// TwinCAT 3 PLC project CarlPlc
// ProgramVersion: 3.1.4022.1
// libraries:
//   Tc2_ModbusRTU, * (Beckhoff Automation GmbH)
//   Tc2_Standard, * (Beckhoff Automation GmbH)
//   Tc2_System, * (Beckhoff Automation GmbH)
//   Tc2_Utilities, * (Beckhoff Automation GmbH)
//   Tc3_Module, * (Beckhoff Automation GmbH)
// project tree:
//   Common/ DetectEvent.TcPOU (not stored), GVL_Common.TcGVL (not stored), TasterEventStates.TcDUT (not stored), TasterEventType.TcDUT (not stored), LinearCalibration.TcDUT (not stored)
//   FlowRateSensor/ GVL_FlowControl.TcGVL, PRG_UpdateFlowRateSensor.TcPOU (not stored)
//   GasAnalysis/ GVL_GasAnalysis.TcGVL (not stored), PRG_GasAnalysis.TcPOU (not stored)
//   GasSupply/ GVL_GasSupply.TcGVL (not stored), PRG_UpdateGasSupply.TcPOU (not stored)
//   MotorControl/ GVL_MotorControl.TcGVL (not stored), PRG_UpdateMotor.TcPOU
//   pHOrpControl/ EN_ModbusReadTarget.TcDUT, GVL_PhOrpControl.TcGVL (not stored), PRG_ReadModbusSensorData.TcPOU, PRG_UpdatePhControl.TcPOU
//   / PlcTask.TcTTO
//   MAIN/ MAIN.TcPOU
//   ReactorPressureControl/ GVL_ReactorPressureControl.TcGVL (not stored), PRG_UpdatePressureSensor.TcPOU (not stored)
//   RoomTempRh/ GVL_TempRHSensor.TcGVL (not stored), PRG_UpdateRoomTempRh.TcPOU
//   TemperatureControl/ EN_TempControlMode.TcDUT (not stored), FB_TON.TcPOU (not stored), GVL_TemperatureControl.TcGVL, FUN_ComputeMovingSetPoint.TcPOU (not stored), PRG_UpdateTemperatureControl.TcPOU (not stored), PRG_BAT_TemperatureControl.TcPOU
//   TemperatureControl/PID/ CLK_PRG.TcPOU (not stored), FB_PWM.TcPOU, FT_DERIV.TcPOU (not stored), FT_PIDWL.TcPOU (not stored), FT_PIWL.TcPOU (not stored), PWM_DC.TcPOU, TP_X.TcPOU (not stored), T_PLC_MS.TcPOU (not stored), T_PLC_US.TcPOU (not stored)
//   TemperatureControl/PID_Hoti/ FT_GET_GAINS.TcPOU, FT_PID_CAS.TcPOU, FT_PID_STERI.TcPOU, FT_P_J.TcPOU
// real-time tasks:
//   TASK PlcTask: cycle T#10ms, priority 20, ADS port 350
// I/O:
//   DEVICE Device 1 (EtherCAT), AmsNetId 5.54.16.198.2.1
//     Term 1 (EK1200) [EK1200-5000 EtherCAT Power supply (2A E-Bus)]
//       Term 2 (EL3014) Motor Speed In [EL3014 4Ch. Ana. Input 0-20mA DIFF]
//       Term 3 (EL4004) Motor Speed Out [EL4004 4Ch. Ana. Output 0-10V, 12bit]
//       Term 4 (EL2004) DO Heating Cooling [EL2004 4Ch. Dig. Output 24V, 0.5A]
//       Term 5 (EL2004) DO Gassing Valves [EL2004 4Ch. Dig. Output 24V, 0.5A]
//       Term 6 (EL2004) DO Motor Control Out [EL2004 4Ch. Dig. Output 24V, 0.5A]
//       Term 7 (EL6021) PhModbus [EL6021 Interface (RS422/485)]
//       Term 8 (EL6021) OrpModbus [EL6021 Interface (RS422/485)]
//       Term 21 (EL1004) DI Gas Analysis [EL1004 4Ch. Dig. Input 24V, 3ms]
//       Term 18 (EL3052) AI Pressure Flow [EL3052 2Ch. Ana. Input 4-20mA]
//       Term 24 (EL3052) AI Heating Cooling [EL3052 2Ch. Ana. Input 4-20mA]
//       Term 10 (EL9184) [EL9184 Potential Connection, 8 x 24V, 8 x Ground]
//       Term 26 (EL3044) [EL3044 4Ch. Ana. Input 0-20mA]
//       Term 9 (EL9011) [EL9011 End Terminal]
// variable links:
//   CarlPlc/CarlPlc Instance <-> Device 1 (EtherCAT)/Term 1 (EK1200)/Term 18 (EL3052) AI Pressure Flow
//     PlcTask Inputs/GVL_FlowControl.flowRateRawCounts <-> FlowRateSensor/FlowRateRaw
//     PlcTask Inputs/GVL_ReactorPressureControl.pressureRawCounts <-> PressureSensor/PressureSensorRaw
//   CarlPlc/CarlPlc Instance <-> Device 1 (EtherCAT)/Term 1 (EK1200)/Term 2 (EL3014) Motor Speed In
//     PlcTask Inputs/GVL_MotorControl.motorActualSpeed <-> AI Motor RPM/Value
//     PlcTask Inputs/GVL_TempRHSensor.roomRhRaw <-> AI Room RH/Value
//     PlcTask Inputs/GVL_TempRHSensor.roomTempRaw <-> AI Room Temp/Value
//   CarlPlc/CarlPlc Instance <-> Device 1 (EtherCAT)/Term 1 (EK1200)/Term 21 (EL1004) DI Gas Analysis
//     PlcTask Inputs/GVL_GasAnalysis.ch4FlowSensor <-> Flow Sensor CH4/Input
//     PlcTask Inputs/GVL_GasAnalysis.o2FlowSensor <-> Flow Sensor O2/Input
//   CarlPlc/CarlPlc Instance <-> Device 1 (EtherCAT)/Term 1 (EK1200)/Term 24 (EL3052) AI Heating Cooling
//     PlcTask Inputs/GVL_TemperatureControl.jacketTempRaw <-> AI Jacket Temp/Value
//   CarlPlc/CarlPlc Instance <-> Device 1 (EtherCAT)/Term 1 (EK1200)/Term 26 (EL3044)
//     PlcTask Inputs/GVL_GasAnalysis.ch4SensorRaw <-> AI CH4/Value
//     PlcTask Inputs/GVL_GasAnalysis.o2SensorRaw <-> AI O2/Value
//     PlcTask Inputs/GVL_GasSupply.gasSupplyPressureRaw <-> AI Gas Supply Pressure/Value
//   CarlPlc/CarlPlc Instance <-> Device 1 (EtherCAT)/Term 1 (EK1200)/Term 3 (EL4004) Motor Speed Out
//     PlcTask Outputs/GVL_MotorControl.motorTargetSpeed <-> MotorTargetSpeed/MotorTargetSpeed
//     PlcTask Outputs/GVL_PhOrpControl.acidPumpSpeedCount <-> AcidPumpSpeedCount/acidPumpSpeedCount
//   CarlPlc/CarlPlc Instance <-> Device 1 (EtherCAT)/Term 1 (EK1200)/Term 4 (EL2004) DO Heating Cooling
//     PlcTask Outputs/GVL_TemperatureControl.coldValve <-> ColdValve/Output
//     PlcTask Outputs/GVL_TemperatureControl.hotValve <-> HotValve/Output
//     PlcTask Outputs/GVL_TemperatureControl.pumpOn <-> PumpOn/Output
//     PlcTask Outputs/GVL_TemperatureControl.steriValve <-> SteriValve/Output
//   CarlPlc/CarlPlc Instance <-> Device 1 (EtherCAT)/Term 1 (EK1200)/Term 5 (EL2004) DO Gassing Valves
//     PlcTask Outputs/GVL_GasSupply.gasSupplyValve <-> GasSupplyValve/Output
//     PlcTask Outputs/GVL_ReactorPressureControl.reactorPressureInletValve <-> reactorPressureInlet/ReactorPressureInlet
//     PlcTask Outputs/GVL_ReactorPressureControl.reactorPressureOutletValve <-> reactorPressureOutlet/Output
//   CarlPlc/CarlPlc Instance <-> Device 1 (EtherCAT)/Term 1 (EK1200)/Term 6 (EL2004) DO Motor Control Out
//     PlcTask Outputs/GVL_MotorControl.motorReset <-> motorReset/Output
//     PlcTask Outputs/GVL_MotorControl.motorStart <-> motorStart/Output
//   CarlPlc/CarlPlc Instance <-> Device 1 (EtherCAT)/Term 1 (EK1200)/Term 7 (EL6021) PhModbus
//     PlcTask Inputs/GVL_Common.PhModbus.InData/D[{0..21}] <-> COM TxPDO-Map Inputs/Data In {0..21}  (22 links)
//     PlcTask Inputs/GVL_Common.PhModbus.InData/Status <-> COM TxPDO-Map Inputs/Status
//     PlcTask Outputs/GVL_Common.PhModbus.OutData/Ctrl <-> COM RxPDO-Map Outputs/Ctrl
//     PlcTask Outputs/GVL_Common.PhModbus.OutData/D[{0..21}] <-> COM RxPDO-Map Outputs/Data Out {0..21}  (22 links)
//   CarlPlc/CarlPlc Instance <-> Device 1 (EtherCAT)/Term 1 (EK1200)/Term 8 (EL6021) OrpModbus
//     PlcTask Inputs/GVL_Common.OrpModbus.InData/D[{0..21}] <-> COM TxPDO-Map Inputs/Data In {0..21}  (22 links)
//     PlcTask Inputs/GVL_Common.OrpModbus.InData/Status <-> COM TxPDO-Map Inputs/Status
//     PlcTask Outputs/GVL_Common.OrpModbus.OutData/Ctrl <-> COM RxPDO-Map Outputs/Ctrl
//     PlcTask Outputs/GVL_Common.OrpModbus.OutData/D[{0..21}] <-> COM RxPDO-Map Outputs/Data Out {0..21}  (22 links)

CONFIGURATION CarlPlc
    RESOURCE PLC ON TwinCAT3
        TASK PlcTask(INTERVAL := T#10ms, PRIORITY := 20);
        PROGRAM MAIN WITH PlcTask : MAIN;
    END_RESOURCE
END_CONFIGURATION

// ---- pHOrpControl/EN_ModbusReadTarget.TcDUT
{attribute 'qualified_only'}
{attribute 'strict'}
TYPE EN_ModbusReadTarget :
(
	READ_TARGET_PH 		:= 1,
	READ_TARGET_PH_T,
	READ_TARGET_ORP,
	READ_TARGET_ORP_T
);
END_TYPE

// ---- FlowRateSensor/GVL_FlowControl.TcGVL
VAR_GLOBAL
	(* flow meter *)
	flowRateRawCounts	AT %I*	: INT := 0;
	flowRateCalibration			: LinearCalibration := (scaleFactor := 8.3415719228868017795353435491844E-5, offset := 0.3);
	flowRateLitersPerMinute		: REAL := 0.0;

	resetSpargeVolume			: BOOL := FALSE;
	resetSpargeVolumeCumulative	: BOOL := FALSE;
	
END_VAR

VAR_GLOBAL PERSISTENT
	spargeVolume 				: REAL;
	spargeVolumeCumulative		: REAL;
END_VAR

// ---- TemperatureControl/GVL_TemperatureControl.TcGVL
VAR_GLOBAL


	tPhCurrent					: REAL := 0.0;
	tPhLastReadingValid			: BOOL := FALSE;
	tOrpCurrent					: REAL := 0.0;
	tOrpLastReadingValid		: BOOL := FALSE;


	(* temperature control *)
	pumpOn				AT %Q* 	: BOOL := FALSE;
	coldValve			AT %Q* 	: BOOL := FALSE;
	hotValve			AT %Q* 	: BOOL := FALSE;
	steriValve			AT %Q*	: BOOL := FALSE; 
	//
	pwmDutyCycle				: REAL := 0.0;	
	
	jacketTempRaw		AT %I*	: INT;
	jacketTempC					: REAL := 0.0;
	jacketTempK					: REAL := 0.0;
	
	
	tempControlStop				: BOOL := FALSE;
	tempControlStart			: BOOL := FALSE;
	hotValveButton				: BOOL := FALSE;
	coldValveButton				: BOOL := FALSE;
	
	pumpIsRunning				: BOOL := FALSE;
	tempControlRunning			: BOOL := FALSE;
	tempSafetyEnabled			: BOOL := FALSE;
	
	steriStart					: BOOL := FALSE;
	steriStop					: BOOL := FALSE;
	steriRunning				: BOOL := FALSE;

	
	currentMeanTemp				: REAL := 0;
	currentTempValid			: BOOL := FALSE;
	(* target temp -> see retains *) 
	
	tempIsBelowSteriTemp		: BOOL := TRUE;
	(* target steri temp --> see retains *)	

	
END_VAR

VAR_GLOBAL PERSISTENT
	targetControlTemp			: REAL;
	targetSteriTemp				: REAL;
	targetSteriTimeMinutes		: INT;
	remainingSteriTimeMinutes	: REAL;
	
	
	remainingSteriTimeInMs		: DINT; (* 30 min in ms *)
	
	countTempSpikes				: INT;
	countValveMaxTimeExceeded	: INT;

	pidResetCounter				: INT;
END_VAR

VAR_GLOBAL CONSTANT
	CYCLE_TIME_IN_MS		: TIME := T#10ms;
END_VAR

// ---- MAIN/MAIN.TcPOU
PROGRAM MAIN
VAR

	
END_VAR

loopCounter := loopCounter + 1;

PRG_ReadModbusSensorData();

(* PRG_HandleUserInputs(); *)

PRG_UpdateMotor();

//PRG_UpdateTemperatureControl();
PRG_BAT_TemperatureControl();

PRG_UpdatePressureSensor();
PRG_UpdateFlowRateSensor();
PRG_UpdatePhControl();
PRG_UpdateGasSupply();
PRG_UpdateRoomTempRh();
PRG_GasAnalysis();

END_PROGRAM

// ---- pHOrpControl/PRG_ReadModbusSensorData.TcPOU
PROGRAM PRG_ReadModbusSensorData
VAR
	
	CurrentReadTarget			: EN_ModbusReadTarget := EN_ModbusReadTarget.READ_TARGET_PH;
	
	ProcessValueRegister		: WORD := 2089;
	TemperatureRegister			: WORD := 2409;
	PhSensorUnitId				: BYTE := 1;
	OrpSensorUnitId				: BYTE := 2;
	RegQuantityToRead			: WORD :=10;
	
	currentUnitId				: BYTE := PhSensorUnitId;
	currentModbusRegister		: WORD := ProcessValueRegister;

	ModbusBusy					: BOOL := FALSE;

	(* diagnostics *)	
	LastModbusError				: ST_ModbusErrorDiagnostics;
	LastErrorstate				: INT;
	CurrentState				: INT;
	CounterError				: INT := 0;
	CounterSuccess				: INT := 0;
	
	firstCall					: BOOL := TRUE;	
	previousCall				: BOOL := FALSE;
	
	scaleFactorPh				: REAL :=   1.210526;
	offsetPh					: REAL := 	-1.231579; 	


	scaleFactorOrp				: REAL := 0.999321727334388;
	offsetOrp					: REAL := 0.0;			
	
END_VAR

(* looping through pH, pH-T, ORP, ORP-T reading the latest values *)
IF firstCall THEN
	PhModbus.ReadRegs( Execute := FALSE);
	OrpModbus.ReadRegs( Execute := FALSE);
	firstCall := FALSE;
	previousCall := TRUE;
END_IF	

CASE  CurrentReadTarget OF 
	EN_ModbusReadTarget.READ_TARGET_PH:
		PhModbus.Readregs (UnitID 		:= PhSensorUnitId ,
   							Quantity   	:= RegQuantityToRead,
   							MBAddr    	:= ProcessValueRegister,
   							cbLength    := RegQuantityToRead*2,
   							pMemoryAddr := ADR(PhValueArrayIn),   
   							Execute    	:= TRUE,
   							Timeout    	:= T#300MS,
							Busy 		=> ModbusBusy	
						  );
		
		IF NOT ModbusBusy THEN
			PhModbus.ReadRegs(Execute:= FALSE);
			CurrentReadTarget := EN_ModbusReadTarget.READ_TARGET_PH_T;
	
			IF PhModbus.Error THEN
				LastModbusError 	:= PhModbus.ErrorDiagnostics;
				LastErrorstate 		:= CurrentState;
				CounterError 		:= CounterError + 1;
				phLastReadingValid 	:= FALSE;
			ELSE
				CounterSuccess 		:= CounterSuccess + 1;
				phLastReadingValid 	:= TRUE;
				phCurrent			:= PhValueArrayIn[1]*scaleFactorPh + offsetPh;
			END_IF
		END_IF
		
	EN_ModbusReadTarget.READ_TARGET_PH_T:
		PhModbus.Readregs (UnitID 		:= PhSensorUnitId ,
   							Quantity   	:= RegQuantityToRead,
   							MBAddr    	:= TemperatureRegister,
   							cbLength    := RegQuantityToRead*2,
   							pMemoryAddr := ADR(TPhValueArrayIn),   
   							Execute    	:= TRUE,
   							Timeout    	:= T#300MS,
							Busy 		=> ModbusBusy	
						  );
		
		IF NOT ModbusBusy THEN
			PhModbus.ReadRegs(Execute:= FALSE);	
			CurrentReadTarget := EN_ModbusReadTarget.READ_TARGET_ORP;

			IF PhModbus.Error THEN
				LastModbusError 	:= PhModbus.ErrorDiagnostics;
				LastErrorstate 		:= CurrentState;
				CounterError 		:= CounterError + 1;
				tPhLastReadingValid := FALSE;
			ELSE
				CounterSuccess 		:= CounterSuccess + 1;
				tPhLastReadingValid := TRUE;
				tPhCurrent			:= TPhValueArrayIn[1];
			END_IF
		END_IF
	
	EN_ModbusReadTarget.READ_TARGET_ORP:
		OrpModbus.Readregs (UnitID 		:= OrpSensorUnitId ,
   							Quantity   	:= RegQuantityToRead,
   							MBAddr    	:= ProcessValueRegister,
   							cbLength    := RegQuantityToRead*2,
   							pMemoryAddr := ADR(OrpValueArrayIn),   
   							Execute    	:= TRUE,
   							Timeout    	:= T#300MS,
							Busy 		=> ModbusBusy	
						  );
		
		IF NOT ModbusBusy THEN
			OrpModbus.ReadRegs(Execute:= FALSE);	
			CurrentReadTarget := EN_ModbusReadTarget.READ_TARGET_ORP_T;

			IF OrpModbus.Error THEN
				LastModbusError 	:= OrpModbus.ErrorDiagnostics;
				LastErrorstate 		:= CurrentState;
				CounterError 		:= CounterError + 1;
				orpLastReadingValid := FALSE;
			ELSE
				CounterSuccess 		:= CounterSuccess + 1;
				orpLastReadingValid := TRUE;
				orpCurrent			:= OrpValueArrayIn[1]*scaleFactorOrp + offsetOrp;
			END_IF
		END_IF

	EN_ModbusReadTarget.READ_TARGET_ORP_T:

		OrpModbus.Readregs (UnitID 		:= OrpSensorUnitId ,
   							Quantity   	:= RegQuantityToRead,
   							MBAddr    	:= TemperatureRegister,
   							cbLength    := RegQuantityToRead*2,
   							pMemoryAddr := ADR(TOrpValueArrayIn),   
   							Execute    	:= TRUE,
   							Timeout    	:= T#300MS,
							Busy 		=> ModbusBusy	
						  );
		
		IF NOT ModbusBusy THEN
			OrpModbus.ReadRegs(Execute:= FALSE);	
			CurrentReadTarget := EN_ModbusReadTarget.READ_TARGET_PH;

			IF OrpModbus.Error THEN
				LastModbusError := OrpModbus.ErrorDiagnostics;
				LastErrorstate 	:= CurrentState;
				CounterError 	:= CounterError + 1;
				tOrpLastReadingValid := FALSE;
			ELSE
				CounterSuccess 	:= CounterSuccess + 1;
				tOrpLastReadingValid := TRUE;
				tOrpCurrent	:= TOrpValueArrayIn[1];
			END_IF
		END_IF
	
END_CASE
			
IF tPhLastReadingValid AND tOrpLastReadingValid THEN
	currentMeanTemp := (tPhCurrent + tOrpCurrent)/2.0;
	currentTempValid := TRUE;
	previousCall := FALSE;
ELSIF tPhLastReadingValid AND NOT tOrpLastReadingValid THEN
	currentMeanTemp := tPhCurrent;
	currentTempValid := TRUE;
	previousCall := FALSE;
ELSIF NOT tPhLastReadingValid AND tOrpLastReadingValid THEN
	currentMeanTemp := tOrpCurrent;
	currentTempValid := TRUE;
	previousCall := FALSE;
ELSE 
	(* no valid temperature signal !! signal to stop temperature control, if active *)
	currentTempValid := FALSE;
	currentMeanTemp := -99.0;	
	tOrpCurrent := -99.0;
	tPhCurrent := -99.0;
	IF firstCall = FALSE AND previousCall = FALSE THEN
		firstCall := TRUE;
	END_IF
END_IF

END_PROGRAM

// ---- MotorControl/PRG_UpdateMotor.TcPOU
PROGRAM PRG_UpdateMotor
VAR
	resetMotor			: RS;
	
	gearingFactor		: INT := 460;
	gearingDivisor		: INT := 6;
	
	motorStartEvt		: DetectEvent;
	motorStopEvt		: DetectEvent;
	
END_VAR

resetMotor(	SET:= motorStartButton, RESET1 := motorStopButton, Q1 => motorStart);
motorTargetSpeed := (currentMotorSpeedSetting * gearingFactor)/gearingDivisor;

motorStartEvt(newSignalValue:= motorStartButton, detectLongClick := FALSE);
motorStopEvt(newSignalValue:= motorStopButton, detectLongClick := FALSE);

IF motorStartEvt.eventDetected = TASTEVT_PositiveEdge THEN
	motorStartButton := FALSE;
END_IF

IF motorStopEvt.eventDetected = TASTEVT_PositiveEdge THEN
	motorStopButton := FALSE;
END_IF

motorRpm := motorActualSpeed*gearingDivisor/gearingFactor;

IF motorStart THEN
	motorRunning := TRUE;
ELSE
	motorRunning := FALSE;
END_IF

(* TODO:
	--> what should happen when "RESET FAILURE" Button is pressed? 
*)

END_PROGRAM

// ---- TemperatureControl/PRG_BAT_TemperatureControl.TcPOU
PROGRAM PRG_BAT_TemperatureControl
VAR
	tempControlMode				: EN_TempControlMode := EN_TempControlMode.TEMP_MODE_MANUAL;  
	
	loopCounter					: DINT := 0;

	(* Controller settings *)
	pwmPeriodinSec			: TIME := T#25S;
	pwmDutyCycle			: REAL := 0.0;	
	pwmOutputValveControl 	: FB_PWM;
	
	//Controling Temperatur for 20°C to 90°C
	CAS_Controller			: FT_PID_CAS;
	
	//Controling Temperatur above 90°C
	STERI_Controller		: FT_PID_STERI;
	
	//GET_GAINS
	GET_GAINS				: FT_GET_GAINS;
	//GAINS JACKET
	kp_J					: REAL ;
	ki_J					: REAL ;
	//GAINS CELL
	kp_C					: REAL ;
	ki_C					: REAL ;
	kd_C					: REAL ;
	
	//Traking time - anti-windup 
	tr_J					: REAL := 1.0;
	tr_C					: REAL := 1.0;
	//is used for changing the status from heating <-> cooling 
	TargetTemp_old 			: REAL ;
	
	// Cooling or Heating for MODE_HEATCOOL;
	COOLING 				: BOOL := FALSE;
	HEATING					: BOOL := FALSE;
		
	errorTemp				: REAL := 0.0;
	pidReset				: BOOL := FALSE;
		
	evtSteriStart			: DetectEvent;
	evtSteriStop			: DetectEvent;
		
	evtTempControlStart		: DetectEvent;
	evtTempControlStop		: DetectEvent;
	
	windUpResetTimer		: TON;
	windUpResetTime			: TIME := T#30S;
	
	maxValveOnTimer		 	: TON;
	maxValveOnTime			: TIME := T#25S;	
	
	evtPidReset				: DetectEvent;
END_VAR

(* jacket temperature input *)
jacketTempC := INT_TO_REAL(jacketTempRaw)/32768.0*200.0 -50.0;
jacketTempK := jacketTempC + 273.15;
tOrpCurrent;
tPhCurrent;
currentMeanTemp;


evtSteriStart(		newSignalValue := steriStart);
evtSteriStop(		newSignalValue := steriStop);
evtTempControlStart(newSignalValue := tempControlStart);
evtTempControlStop(	newSignalValue := tempControlStop);
evtPidReset( 		newSignalValue := pidReset);


IF evtSteriStart.eventDetected = TASTEVT_PositiveEdge THEN
	steriStart := FALSE;
	pumpOn := FALSE;
	CAS_Controller( RST:= TRUE );
	STERI_Controller(RST:=TRUE);
	tempControlMode	:= EN_TempControlMode.TEMP_MODE_STERI;
	tempControlRunning := FALSE;
	steriRunning := TRUE;
	steriValve := FALSE;
	coldValve := FALSE;
	hotValve := FALSE;
	(* Set remaining steri temp *)
	remainingSteriTimeInMs := targetSteriTimeMinutes*60*1000; 
END_IF

IF evtTempControlStart.eventDetected = TASTEVT_PositiveEdge THEN
	tempControlStart := FALSE;
	pumpOn := FALSE;
	CAS_Controller( RST:= TRUE );
	STERI_Controller(RST:=TRUE);
	tempControlMode	:= EN_TempControlMode.TEMP_MODE_HEATCOOL;
	tempControlRunning := TRUE;
	steriRunning := FALSE;
	steriValve := FALSE;
	coldValve := FALSE;
	hotValve := FALSE;
END_IF

IF 	evtSteriStop.eventDetected = TASTEVT_PositiveEdge OR
 	evtTempControlStop.eventDetected = TASTEVT_PositiveEdge 
THEN
	steriStop := FALSE;
	tempControlStop := FALSE;
	pumpOn := FALSE;
	CAS_Controller( RST:= TRUE );
	STERI_Controller(RST:=TRUE);
	tempControlRunning := FALSE;
	steriRunning := FALSE;
	tempControlMode	:= EN_TempControlMode.TEMP_MODE_MANUAL;
	coldValve := FALSE;
	hotValve := FALSE;
	steriValve := FALSE;
	(* TODO: Reset Steri Timer *)
END_IF

(* check if current temperature reading actually valid, otherwise stop any type of temperature control *)

IF NOT currentTempValid THEN
	tempControlMode := EN_TempControlMode.TEMP_MODE_MANUAL;
END_IF


CASE tempControlMode OF
	EN_TempControlMode.TEMP_MODE_MANUAL:
		pumpOn := FALSE;
		CAS_Controller( RST:= TRUE );
		STERI_Controller(RST:=TRUE);
		coldValve := FALSE;
		hotValve := FALSE;
		steriValve := FALSE;
		
		
	EN_TempControlMode.TEMP_MODE_HEATCOOL:
		
		pumpOn := TRUE;
		(* errorTemp := targetControlTemp - currentMeanTemp; *)
		errorTemp := FUN_ComputeMovingSetPoint(currentTemp := currentMeanTemp, targetSetPoint := targetControlTemp) - currentMeanTemp;
		
		//Setting Heating or Cooling only when TargetTemp is changed or ...
		// 	...	errorTemp is lower than 2 Degree so it changes to heating - has to be adjusted
		IF TargetTemp_old = targetControlTemp THEN
			;
			ELSE
				//-----COOLING-----
			IF (TargetTemp_old > targetControlTemp) AND (targetControlTemp <40) AND (errorTemp > 2) THEN
				COOLING := TRUE;
				HEATING := FALSE;
				GET_GAINS( 	TEMP := targetControlTemp,
							MODE := 0,);
				kp_J := GET_GAINS.K_P_J;
				ki_J := GET_GAINS.K_I_J;
				tr_J := GET_GAINS.T_R_J;
 				kp_C := GET_GAINS.K_P_C;
				ki_C := GET_GAINS.K_I_C;
				kd_C := GET_GAINS.K_D_C;
				tr_C := GET_GAINS.T_R_C;
				//-----HEATING-----
			ELSE
				COOLING := FALSE;
				HEATING := TRUE;	
				GET_GAINS( 	TEMP := targetControlTemp,
							MODE := 1,);
				kp_J := GET_GAINS.K_P_J;
				ki_J := GET_GAINS.K_I_J;
				tr_J := GET_GAINS.T_R_J;
 				kp_C := GET_GAINS.K_P_C;
				ki_C := GET_GAINS.K_I_C;
				kd_C := GET_GAINS.K_D_C;
				tr_C := GET_GAINS.T_R_C;
			END_IF
		END_IF
		//Save old TargetTemp
		TargetTemp_old := TargetControlTemp;	 
		//Start Temp. Controller
		CAS_Controller(	T_ERR_C := errorTemp,		//Cell Temperatur error 
						K_P_J 	:= kp_J,
						K_I_J 	:= ki_J,
						T_R_J 	:= tr_J,
						K_P_C 	:= kp_C,	
						K_I_C 	:= ki_C,
						K_D_C 	:= kd_C,			
						T_R_C	:= tr_C, 			//Tracking time used for Anti-Wind up
						T_R_J	:= tr_J,			//Tracking time used for Anti-Wind up
						LIM_L 	:= 0.0,				//Min. Temp for Jacket
						LIM_H 	:= 90.0,			//Max. Temp for Jacket
						RST 	:= pidReset,
						);
												
		pwmDutyCycle := CAS_Controller.P_J_Controll.Y; (* !! pwm block cannot handle negative inputs *)
		//pwmDutyCycle := 1;

		pwmOutputValveControl(pwmCycleTime:=pwmPeriodinSec, pwmDutyCycle:=pwmDutyCycle);	
						
		IF  HEATING = TRUE THEN			 	//heating 
			coldValve := FALSE;
			hotValve := pwmOutputValveControl.Q;
			steriValve := FALSE;
			
		ELSIF COOLING = TRUE THEN			//cooling 
			coldValve := pwmOutputValveControl.Q;
			hotValve := FALSE;
			steriValve := FALSE;
			
		ELSE								//ERROR STATE?
			coldValve := FALSE;
			hotValve := FALSE;
			steriValve := FALSE;
		END_IF
		
//----------------------------------------------STERIL-------------------------------------------------------------------			
	EN_TempControlMode.TEMP_MODE_STERI:
		pumpOn := FALSE;
		errorTemp := targetSteriTemp - currentMeanTemp;
		
		//Setting Heating or Cooling only when TargetTemp is changed
		IF TargetTemp_old = targetControlTemp THEN
			;
			ELSE
			IF (TargetTemp_old > targetControlTemp) THEN
				COOLING := FALSE;
				HEATING := FALSE;

			ELSE
				COOLING := FALSE;
				HEATING := TRUE;	
				GET_GAINS( 	TEMP := targetControlTemp,
							MODE := 0,);
				kp_C := GET_GAINS.K_P_C;
				ki_C := GET_GAINS.K_I_C;
				kd_C := GET_GAINS.K_D_C;
				tr_C := GET_GAINS.T_R_C;
			END_IF
		END_IF
		//Save old TargetTemp
		TargetTemp_old := TargetControlTemp;	
		//Start Temp. Controller
		STERI_Controller(	
						T_ERR_C := errorTemp,		//Cell Temperatur error 
						K_P_C 	:= kp_C,	
						K_I_C 	:= ki_C,
						K_D_C 	:= kd_C,			
						T_R_C	:= tr_C, 			//Tracking time used for Anti-Wind up
						LIM_L 	:= 0.0,				//Min. Temp for Jacket
						LIM_H 	:= 1.0,				//Max. Temp for Jacket
						RST 	:= pidReset,
						);
						
		pwmDutyCycle := STERI_Controller.Y; 	
		//pwmDutyCycle := 0.5;
		
		pwmOutputValveControl(pwmCycleTime:=pwmPeriodinSec, pwmDutyCycle:=pwmDutyCycle);
				
		IF HEATING = TRUE THEN
			(* heating *)
			coldValve 	:= FALSE;
			steriValve 	:= pwmOutputValveControl.Q;
			hotValve 	:= FALSE;
			
		ELSE
			(* cooling *)
			steriValve 	:= FALSE;
			hotValve 	:= FALSE;			
		END_IF
		
		IF currentMeanTemp > (targetSteriTemp-0.5) THEN
			(* count down 10 ms each cycle *)
			remainingSteriTimeInMs := remainingSteriTimeInMs - 10;
			IF remainingSteriTimeInMs < 0 THEN
				tempControlMode := EN_TempControlMode.TEMP_MODE_MANUAL;
				steriValve := FALSE;
				coldValve := FALSE;
				steriStop := TRUE;
			END_IF
		END_IF		
		remainingSteriTimeMinutes := DINT_TO_REAL(remainingSteriTimeInMs)/(60.0*1000.0);
	
	
END_CASE
 
IF evtPidReset.eventDetected = TASTEVT_PositiveEdge THEN
	pidReset := FALSE;
	CAS_Controller(RST:=TRUE);
	STERI_Controller(RST:=TRUE);
	pidResetCounter := pidResetCounter + 1;
	steriValve := FALSE;
	coldValve := FALSE;
	hotValve := FALSE;
END_IF

END_PROGRAM

// ---- TemperatureControl/PID/FB_PWM.TcPOU
FUNCTION_BLOCK FB_PWM
VAR_INPUT
	pwmCycleTime 		: TIME := T#10S;
	pwmDutyCycle		: REAL := 0.5;
	reset				: BOOL := FALSE;
END_VAR
VAR_OUTPUT
	Q					: BOOL := FALSE;
END_VAR
VAR
	pwmTimeInMs			: REAL	:= 0;
	pwmTimer			: FB_TON;
	dutyCycleInMs		: TIME;
	test				: INT;
	internalReset 		: BOOL := FALSE;
	goHigh				: BOOL := FALSE;
	
	temp1				: REAL;
	temp2				: DINT;
	temp3				: REAL;
	temp4				: REAL;
	
END_VAR

IF pwmDutyCycle < 0 THEN
	pwmDutyCycle := 0.0;
END_IF

IF reset OR internalReset THEN
	pwmTimer(IN:= FALSE);
	reset := FALSE;
	internalReset := FALSE;
	IF goHigh THEN
		temp1 := (1.0-pwmDutyCycle);
		temp2 := REAL_TO_DINT(pwmTimeInMs*(1.0-pwmDutyCycle));
		dutyCycleInMs := DINT_TO_TIME(REAL_TO_DINT(pwmTimeInMs*(1.0-pwmDutyCycle)));
		goHigh := FALSE;
	ELSE
		temp1 := (1.0-pwmDutyCycle);
		temp2 := REAL_TO_DINT(pwmTimeInMs*(1.0-pwmDutyCycle));
		dutyCycleInMs := DINT_TO_TIME(REAL_TO_DINT(pwmTimeInMs*pwmDutyCycle));
	END_IF
ELSE
	pwmTimeInMs := DINT_TO_REAL(TIME_TO_DINT(pwmCycleTime));
	IF Q THEN
		(* high  --> running falling timer *)
		(*dutyCycleInMs := DINT_TO_TIME(REAL_TO_DINT(pwmTimeInMs*pwmDutyCycle));*)
		pwmTimer(IN:=TRUE, PT:=dutyCycleInMs);
		IF pwmTimer.Q THEN
			internalReset := TRUE;
			Q := FALSE;
			goHigh := TRUE;
			pwmTimer(IN:=FALSE);
		END_IF		
	ELSE
		(* low --> running rising timer *)
		pwmTimer(IN:=TRUE, PT:=dutyCycleInMs);
		IF pwmTimer.Q THEN
			internalReset := TRUE;
			Q := TRUE;
			pwmTimer(IN:=FALSE);
		END_IF		
	END_IF
END_IF

END_FUNCTION_BLOCK

// ---- TemperatureControl/PID_Hoti/FT_PID_CAS.TcPOU
FUNCTION_BLOCK FT_PID_CAS
VAR_INPUT
	T_ERR_C	: REAL;					//Error
	MODE 	: BOOL;
	//Jacket
	K_P_J 	: REAL := 1.0; 
	K_I_J	: REAL := 1.0;	
	// Cell
	K_P_C 	: REAL := 1.0;		
	K_I_C 	: REAL := 1.0;
	K_D_C 	: REAL := 1.0;
	T_R_C	: REAL := 1.0; 			//Tracking time used for Anti-Wind up
	T_R_J	: REAL := 1.0; 			//Tracking time used for Anti-Wind up
	LIM_L 	: REAL := -1.0E38;		//Min. Temp for Jacket
	LIM_H 	: REAL := 1.0E38;		//Max. Temp for Jacket
	RST 	: BOOL;
END_VAR
VAR_OUTPUT
	Y 		: REAL;
	LIM 	: BOOL;
END_VAR
VAR
	//For Cell
	P_C 	: REAL;			//Proportional term
	I_C 	: REAL;			//Integral term
	D_C 	: REAL;			//Derivate term
	err_sum : REAL :=0;		//error for I
	err_k_1 : REAL :=0;		//old error
	
	//for the jacket
	P_J 	: REAL :=1.0;
	
	//Control for Jacket
	J_Controll : FT_P_J ;
	
	oldMode : BOOL;
	
	//Saturation
	y_k		: REAL;			//control signal 
	y_sat   : REAL;			//Control signal after saturation
	y_k_1 	: REAL;			//Control signal (k-1)
	y_sat_k_1 :REAL;		//control signal after saturation (k-1)
	
	I_C_k_1	: REAL ; 		//I-Part old
	
	T_ERR_J : REAL ;			
	T_ERR_J_N : REAL ;	
	
	tx		: DWORD;
	T_a		: REAL := 0.01;			//Sampling Time
	t_last	: DWORD;
END_VAR

(* if rst then *)
IF rst THEN		//Reset -- tbd
	err_sum:=0;
	err_k_1:=0;
	t_last := T_PLC_US();
	T_a := 0.010;
	I_C :=0;
	D_C :=0;
ELSE
	//read last cycle time in Microseconds
	tx := T_PLC_US();
	T_a := DWORD_TO_REAL(tx - t_last)/1000000;
	t_last := tx;
	
	IF (MODE = TRUE) THEN
		T_ERR_C:=(T_ERR_C*-1);	
	END_IF
	
	IF (oldMode <> MODE) THEN
		I_C_k_1 := 0;
	END_IF
	
	//proportional term
	P_C := K_P_C*T_ERR_C;
	
	//Integrator term with Anti-Windup backcalculation
	err_sum:=err_k_1+T_ERR_C;
	I_C := I_C_k_1 + K_I_C * err_sum * T_a/2.0 + //(T_a/T_R_C)*(y_sat-y_k);
	
	//Derivative term
	//D_C := K_D_C * (T_ERR_C-err_k_1);//T_a;
	
	//output before saturation
	y_k := P_C + I_C + D_C;
	
	//Saturation used to limit Jacket temp.
	IF LIM_H < y_k THEN
		y_sat:= LIM_H;
	ELSIF  LIM_L > y_k THEN
		y_sat:= LIM_L;
	ELSE
		y_sat:= y_k;
	END_IF	
	
	//setting output
	Y	:= y_sat;	
	
	IF (MODE = TRUE) THEN
		T_ERR_J :=jacketTempC -Y;	
	ELSE
		//Jacket ERROR
		T_ERR_J := Y - jacketTempC;	
	END_IF	
	
	oldMode:= MODE;
	
	//IF (MODE = TRUE) THEN
	//T_ERR_J:=(T_ERR_J*-1);	
	//END_IF
	
	//Jacket Controll
	J_Controll (	T_ERR_J := T_ERR_J, 
					K_P_J := K_P_J,
					K_I_J := K_I_J,
					T_R_J := T_R_J,
					RST := RST,
					);
					
	//save variable for next step
	I_C_k_1 := I_C;			//Saving Integral part for next step
	err_k_1 := T_ERR_C;			//Saving error for ...
END_IF

END_FUNCTION_BLOCK

// ---- TemperatureControl/PID_Hoti/FT_P_J.TcPOU
FUNCTION_BLOCK FT_P_J
VAR_INPUT
	T_ERR_J	: REAL;					//Error
	K_P_J	: REAL;
	K_I_J	: REAL;
	T_R_J	: REAL; 				//Tracking time used for Anti-Wind up
	RST 	: BOOL;
END_VAR
VAR_OUTPUT
	Y 		: REAL;
END_VAR
VAR
	P_J 	: REAL;	
	I_J		: REAL;
	err_sum	: REAL;
	err_k_1 : REAL;
	I_J_k_1 : REAL;
	
	//Max min PWM 0..1;
	LIM_L 	: REAL :=0.0;	
	LIM_H	: REAL :=1.0;
	
	//Saturation
	y_k		: REAL;			//control signal 
	y_sat   : REAL;			//Control signal after saturation
	y_k_1 	: REAL;			//Control signal (k-1)
	y_sat_k_1 :REAL;		//control signal after saturation (k-1)
	
	I_C_k_1 : REAL;			//I-Part old
	
	tx		: DWORD;
	T_a		: REAL;			//Sampling Time
	t_last	: DWORD;
END_VAR

IF rst THEN		//Reset -- tbd
	err_sum:=0;
	err_k_1:=0;
	t_last := T_PLC_US();
	T_a := 0.0;
ELSE
	tx := T_PLC_US();
	T_a := DWORD_TO_REAL(tx - t_last);
	t_last := tx;
	
	//proportional term
	P_J := K_P_J*T_ERR_J;
	
	//if necessary - integral term
	(*
	err_sum:=err_k_1+T_ERR_J;
	I_J := I_J_k_1 + K_I_J * err_sum * T_a/2.0 + (T_a/T_R_J)*(y_k-y_sat+y_k_1-y_sat_k_1);		
	*)
	
	I_J :=0;				//if Integral in use --> delete this part------!!!!
	
	//output before saturation
	y_k := P_J + I_J ;
	
	//Saturation used to limit Jacket temp.
	IF LIM_H < y_k THEN
		y_sat:= LIM_H;
	ELSIF  LIM_L > y_k THEN
		y_sat:= LIM_L;
	ELSE
		y_sat:= y_k;
	END_IF	
	
	//setting output
	Y := y_sat;
	
	//save variable for next step
	I_J_k_1 := I_J;			//Saving Integral part for next step
END_IF

END_FUNCTION_BLOCK

// ---- TemperatureControl/PID_Hoti/FT_PID_STERI.TcPOU
FUNCTION_BLOCK FT_PID_STERI
VAR_INPUT
	T_ERR_C	: REAL;					//Error
	// Cell
	K_P_C 	: REAL := 1.0;		
	K_I_C 	: REAL := 1.0;
	K_D_C 	: REAL := 1.0;
	T_R_C	: REAL := 1.0; 			//Tracking time used for Anti-Wind up
	LIM_L 	: REAL := 0.0;			//Min. PWM
	LIM_H 	: REAL := 1.0;			//Max. PWM
	RST 	: BOOL;
END_VAR
VAR_OUTPUT
	Y 		: REAL;
	LIM 	: BOOL;
END_VAR
VAR
	//For Cell
	P_C 	: REAL;			//Proportional term
	I_C 	: REAL;			//Integral term
	D_C 	: REAL;			//Derivate term
	err_sum : REAL :=0;		//error for I
	err_k_1 : REAL :=0;		//old error
	
	
	//Saturation
	y_k		: REAL;			//control signal 
	y_sat   : REAL;			//Control signal after saturation
	y_k_1 	: REAL;			//Control signal (k-1)
	y_sat_k_1 :REAL;		//control signal after saturation (k-1)
	
	I_C_k_1	: REAL ; 		//I-Part old
	
	tx		: DWORD;
	T_a		: REAL;			//Sampling Time
	t_last	: DWORD;
END_VAR

(* if rst then *)
IF rst THEN		//Reset -- tbd
	err_sum:=0;
	err_k_1:=0;
	t_last := T_PLC_US();
	T_a := 0.0;
ELSE
	//read last cycle time in Microseconds
	tx := T_PLC_US();
	T_a := DWORD_TO_REAL(tx - t_last);
	t_last := tx;
	
	//proportional term
	P_C := K_P_C*T_ERR_C;
	
	//Integrator term with Anti-Windup backcalculation
	err_sum:=err_k_1+T_ERR_C;
	I_C := I_C_k_1 + K_I_C * err_sum * T_a/2.0 + (T_a/T_R_C)*(y_k-y_sat+y_k_1-y_sat_k_1);
	
	//Derivative term
	D_C := K_D_C * (T_ERR_C-err_k_1)/T_a;
	
	//output before saturation
	y_k := P_C + I_C + D_C;
	
	//Saturation used to limit Jacket temp.
	IF LIM_H < y_k THEN
		y_sat:= LIM_H;
	ELSIF  LIM_L > y_k THEN
		y_sat:= LIM_L;
	ELSE
		y_sat:= y_k;
	END_IF	
	
	//setting output
	Y	:= y_sat;	
	
	//save variable for next step
	I_C_k_1 := I_C;				//Saving Integral part for next step
	err_k_1 := T_ERR_C;			//Saving error for ...
END_IF

END_FUNCTION_BLOCK

// ---- TemperatureControl/PID_Hoti/FT_GET_GAINS.TcPOU
FUNCTION_BLOCK FT_GET_GAINS
VAR_INPUT
	TEMP 	: REAL;
	MODE	: BOOL;		// COOLING =0 ; HEATING = 1
END_VAR
VAR_OUTPUT
	//Jacket
	K_P_J 	: REAL;
	K_I_J	: REAL; 
	// Cell
	K_P_C 	: REAL ;		
	K_I_C 	: REAL ;
	K_D_C 	: REAL ;
	//Tracking time 
	T_R_C	: REAL ; 			
	T_R_J	: REAL ; 			
END_VAR
VAR
	TempCase : INT;
END_VAR

IF MODE= TRUE THEN			//HEATING
	IF TEMP < 40 THEN
		TempCase := 1 ;		// 37°C 
	ELSIF TEMP <71 THEN
		TempCase := 2 ;		// up to 71°C 
	ELSIF TEMP <81 THEN
		TempCase := 3 ;		// up to 81°C 
	ELSIF TEMP <91 THEN				
		TempCase := 3 ;		// up to 91°C 
	ELSIF TEMP >115 THEN
		TempCase := 5 ;		// for 121°C
	ELSE
		TempCase := 4 ;		// if over 90°C and below 115 it will handle like 90°C 
	END_IF
ELSE
		TempCase := 0;
END_IF 

CASE TempCase  OF
0:	//COOLING --- till 40°C
	K_P_J := 10;
	K_I_J := 1;
	T_R_J := 1;
	
	K_P_C := 7;
	K_I_C := 0.0021;
	K_D_C := 1050;	
	T_R_C := 714;	
1:  // HEATING ---for 37°C 
	K_P_J := 10;
	K_I_J := 1;
	T_R_J := 1;
	
	K_P_C := 182.5;
	K_I_C := 0.162;
	K_D_C := 385.9;	
	T_R_C := 48.77;	
2:	// HEATING ---for 71°C 
	K_P_J := 10;
	K_I_J := 1;
	T_R_J := 1;
	
	K_P_C := 182.5;
	K_I_C := 0.162;
	K_D_C := 385.9;	
	T_R_C := 48.77;
3:	// HEATING ---for 81°C 
	K_P_J := 10;
	K_I_J := 1;
	T_R_J := 1;
	
	K_P_C := 107.27;
	K_I_C := 0.128;
	K_D_C := 268.18;	
	T_R_C := 45.65;	
4:	// HEATING --- for 91°C  ----tbd
	K_P_J := 1;
	K_I_J := 1;
	T_R_J := 1;
	
	K_P_C := 1;
	K_I_C := 1;
	K_D_C := 1;	
	T_R_C := 1;	
5:	// STERIL --- for 121°C 

	K_P_C := 0.13;
	K_I_C := 0.0000349;
	K_D_C := 9.28;	
	T_R_C := 515.5;	
END_CASE

END_FUNCTION_BLOCK

// ---- pHOrpControl/PRG_UpdatePhControl.TcPOU
PROGRAM PRG_UpdatePhControl
VAR
	evtPhControlStart		: DetectEvent;
	evtPhControlStop		: DetectEvent;
	
END_VAR

evtPhControlStart(newSignalValue := phStart);
evtPhControlStop(newSignalValue := phStop);

IF evtPhControlStart.eventDetected = TASTEVT_PositiveEdge THEN
	phRunning := TRUE;
END_IF

IF evtPhControlStop.eventDetected = TASTEVT_PositiveEdge THEN
	phRunning := FALSE;
END_IF

IF pressureBar < 0.5 AND pressureBar > 0 AND phPumpManual THEN
	acidPumpSpeedCount := REAL_TO_INT(INT_TO_REAL(acidPumpSpeedSetting)*acidPumpSpeedCalibration.scaleFactor + acidPumpSpeedCalibration.offset);
	phPumpRunning := TRUE;
ELSE
	acidPumpSpeedCount := 0;
	phPumpRunning := FALSE;
END_IF

END_PROGRAM

// ---- RoomTempRh/PRG_UpdateRoomTempRh.TcPOU
PROGRAM PRG_UpdateRoomTempRh
VAR
END_VAR

(* currently on 0-20mA inputs, but delivering 4-20mA --> need remove 4mA from Signal *)

roomTemp := (INT_TO_REAL(roomTempRaw)/32767.0)*100.0 - 40.0;  (* Sensor Range: -40°C to + 60°C *)
roomRh :=   (INT_TO_REAL(roomRhRaw)/32767.0)*100.0;

END_PROGRAM

// ---- TemperatureControl/PID/PWM_DC.TcPOU
FUNCTION_BLOCK PWM_DC
VAR_INPUT
	F : REAL;
	DC : REAL;
END_VAR
VAR_OUTPUT
	Q : BOOL;
END_VAR
VAR
	clk: CLK_PRG;
	pulse: TP_X;
	tmp: REAL;
END_VAR

(*this signal generator generates a square wave signal which is specified by the frequency and the duty cycle
*)

IF F > 0.0 THEN
	tmp := 1000.0 / F;
	CLK(PT := REAL_TO_TIME(tmp));
	Pulse(in := clk.Q, pt := REAL_TO_TIME(tmp * DC));
	Q := pulse.Q;
END_IF;

END_FUNCTION_BLOCK
